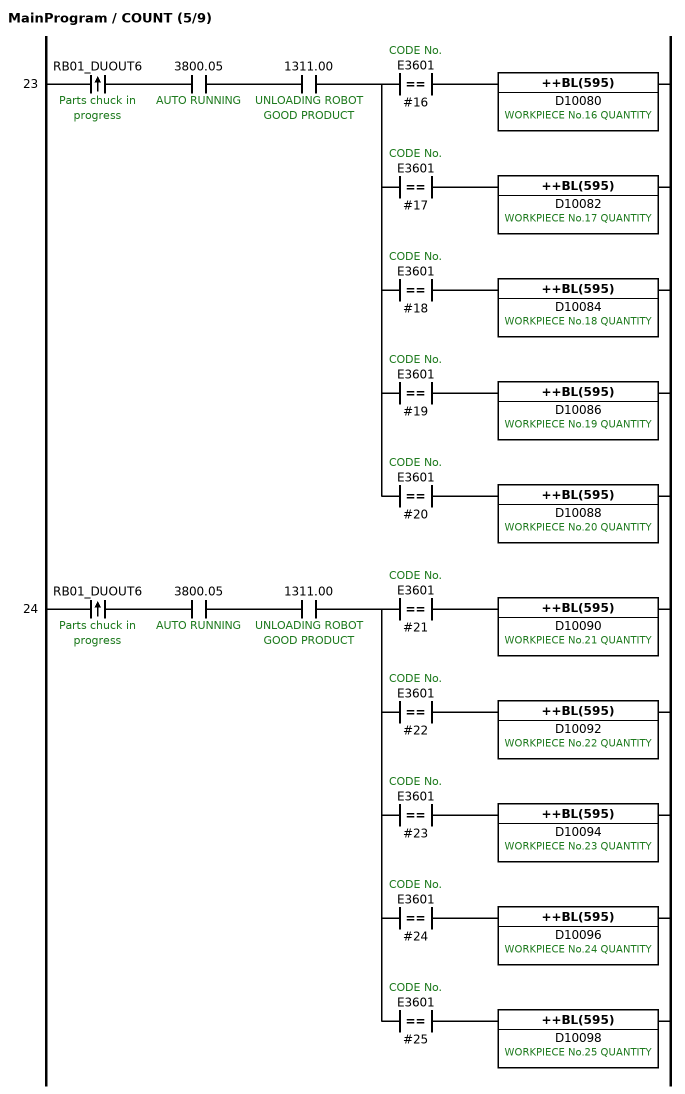
; [picture p144: MainProgram / COUNT, rungs 23-24]
; rung 23
@LD RB01_DUOUT6  ; Parts chuck in progress
AND 3800.05  ; AUTO RUNNING
AND 1311.00  ; UNLOADING ROBOT GOOD PRODUCT
OUT TR0
AND=(300) E3601 #16  ; CODE No.
++BL(595) D10080  ; WORKPIECE No.16 QUANTITY
LD TR0
AND=(300) E3601 #17  ; CODE No.
++BL(595) D10082  ; WORKPIECE No.17 QUANTITY
LD TR0
AND=(300) E3601 #18  ; CODE No.
++BL(595) D10084  ; WORKPIECE No.18 QUANTITY
LD TR0
AND=(300) E3601 #19  ; CODE No.
++BL(595) D10086  ; WORKPIECE No.19 QUANTITY
LD TR0
AND=(300) E3601 #20  ; CODE No.
++BL(595) D10088  ; WORKPIECE No.20 QUANTITY
; rung 24
@LD RB01_DUOUT6  ; Parts chuck in progress
AND 3800.05  ; AUTO RUNNING
AND 1311.00  ; UNLOADING ROBOT GOOD PRODUCT
OUT TR0
AND=(300) E3601 #21  ; CODE No.
++BL(595) D10090  ; WORKPIECE No.21 QUANTITY
LD TR0
AND=(300) E3601 #22  ; CODE No.
++BL(595) D10092  ; WORKPIECE No.22 QUANTITY
LD TR0
AND=(300) E3601 #23  ; CODE No.
++BL(595) D10094  ; WORKPIECE No.23 QUANTITY
LD TR0
AND=(300) E3601 #24  ; CODE No.
++BL(595) D10096  ; WORKPIECE No.24 QUANTITY
LD TR0
AND=(300) E3601 #25  ; CODE No.
++BL(595) D10098  ; WORKPIECE No.25 QUANTITY

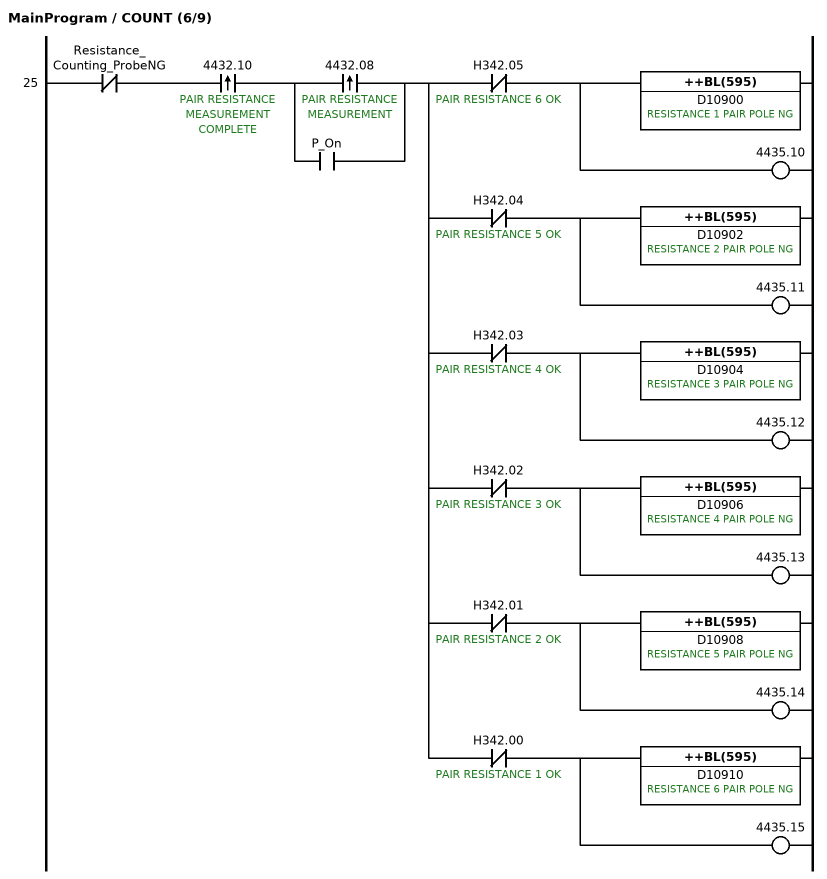
; rung 25
LDNOT Resistance_Counting_ProbeNG
@AND 4432.10  ; PAIR RESISTANCE MEASUREMENT COMPLETE
@LD 4432.08  ; PAIR RESISTANCE MEASUREMENT
OR P_On
ANDLD
OUT TR0
ANDNOT H342.05  ; PAIR RESISTANCE 6 OK
++BL(595) D10900  ; RESISTANCE 1 PAIR POLE NG
OUT 4435.10
LD TR0
ANDNOT H342.04  ; PAIR RESISTANCE 5 OK
++BL(595) D10902  ; RESISTANCE 2 PAIR POLE NG
OUT 4435.11
LD TR0
ANDNOT H342.03  ; PAIR RESISTANCE 4 OK
++BL(595) D10904  ; RESISTANCE 3 PAIR POLE NG
OUT 4435.12
LD TR0
ANDNOT H342.02  ; PAIR RESISTANCE 3 OK
++BL(595) D10906  ; RESISTANCE 4 PAIR POLE NG
OUT 4435.13
LD TR0
ANDNOT H342.01  ; PAIR RESISTANCE 2 OK
++BL(595) D10908  ; RESISTANCE 5 PAIR POLE NG
OUT 4435.14
LD TR0
ANDNOT H342.00  ; PAIR RESISTANCE 1 OK
++BL(595) D10910  ; RESISTANCE 6 PAIR POLE NG
OUT 4435.15

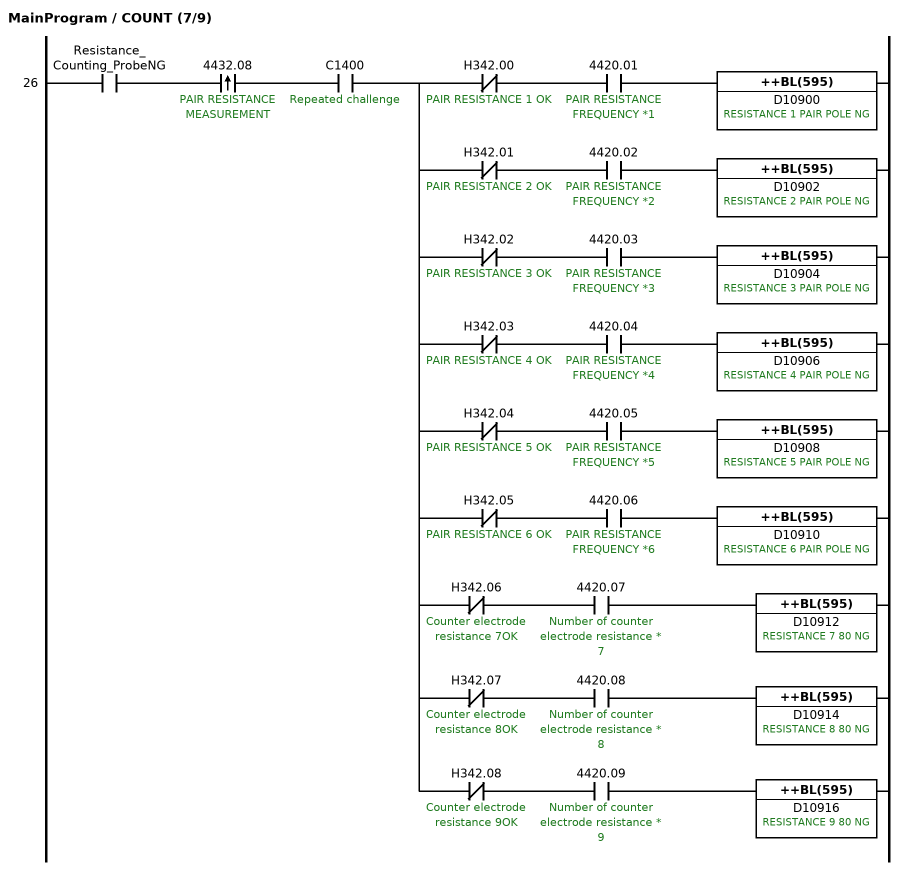
; rung 26
LD Resistance_Counting_ProbeNG
@AND 4432.08  ; PAIR RESISTANCE MEASUREMENT
AND C1400  ; Repeated challenge
OUT TR0
ANDNOT H342.00  ; PAIR RESISTANCE 1 OK
AND 4420.01  ; PAIR RESISTANCE FREQUENCY *1
++BL(595) D10900  ; RESISTANCE 1 PAIR POLE NG
LD TR0
ANDNOT H342.01  ; PAIR RESISTANCE 2 OK
AND 4420.02  ; PAIR RESISTANCE FREQUENCY *2
++BL(595) D10902  ; RESISTANCE 2 PAIR POLE NG
LD TR0
ANDNOT H342.02  ; PAIR RESISTANCE 3 OK
AND 4420.03  ; PAIR RESISTANCE FREQUENCY *3
++BL(595) D10904  ; RESISTANCE 3 PAIR POLE NG
LD TR0
ANDNOT H342.03  ; PAIR RESISTANCE 4 OK
AND 4420.04  ; PAIR RESISTANCE FREQUENCY *4
++BL(595) D10906  ; RESISTANCE 4 PAIR POLE NG
LD TR0
ANDNOT H342.04  ; PAIR RESISTANCE 5 OK
AND 4420.05  ; PAIR RESISTANCE FREQUENCY *5
++BL(595) D10908  ; RESISTANCE 5 PAIR POLE NG
LD TR0
ANDNOT H342.05  ; PAIR RESISTANCE 6 OK
AND 4420.06  ; PAIR RESISTANCE FREQUENCY *6
++BL(595) D10910  ; RESISTANCE 6 PAIR POLE NG
LD TR0
ANDNOT H342.06  ; Counter electrode resistance 7OK
AND 4420.07  ; Number of counter electrode resistance * 7
++BL(595) D10912  ; RESISTANCE 7 80 NG
LD TR0
ANDNOT H342.07  ; Counter electrode resistance 8OK
AND 4420.08  ; Number of counter electrode resistance * 8
++BL(595) D10914  ; RESISTANCE 8 80 NG
LD TR0
ANDNOT H342.08  ; Counter electrode resistance 9OK
AND 4420.09  ; Number of counter electrode resistance * 9
++BL(595) D10916  ; RESISTANCE 9 80 NG

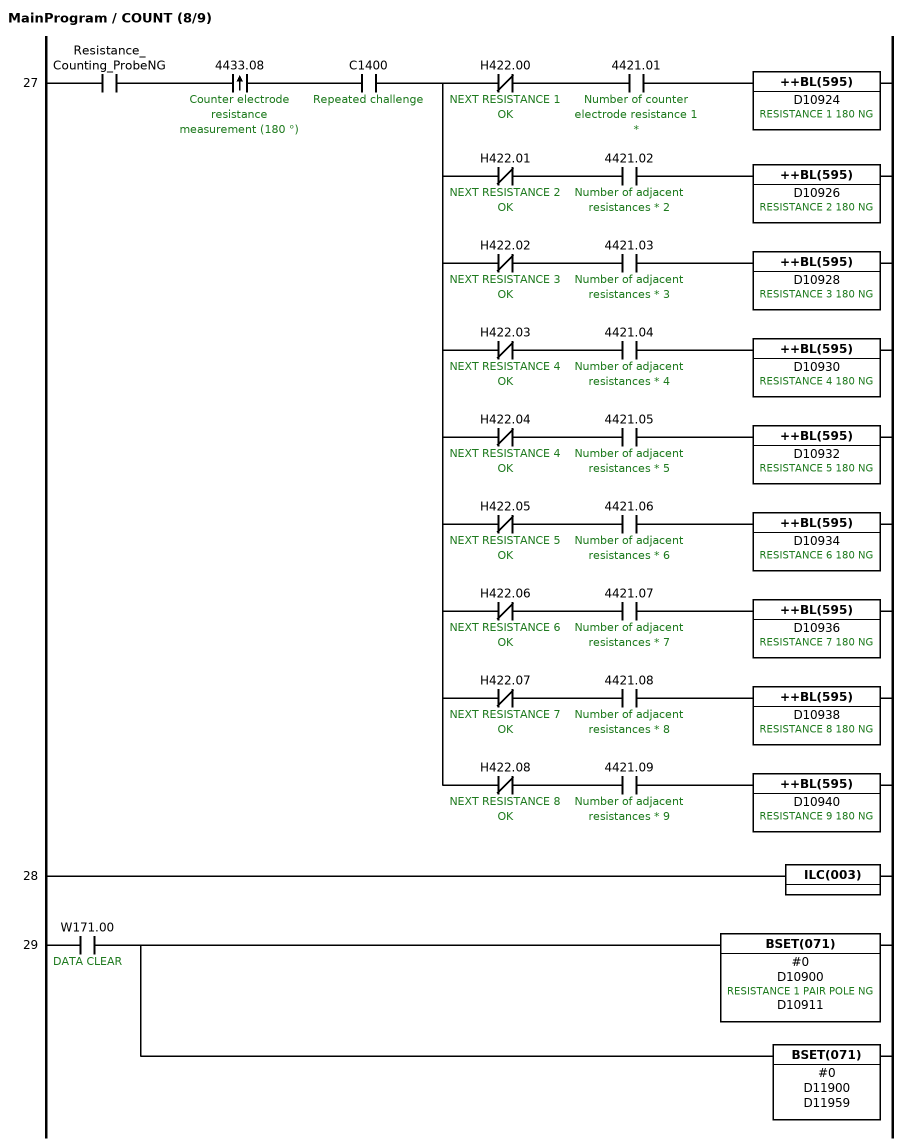
; rung 27
LD Resistance_Counting_ProbeNG
@AND 4433.08  ; Counter electrode resistance measurement (180 °)
AND C1400  ; Repeated challenge
OUT TR0
ANDNOT H422.00  ; NEXT RESISTANCE 1 OK
AND 4421.01  ; Number of counter electrode resistance 1 *
++BL(595) D10924  ; RESISTANCE 1 180 NG
LD TR0
ANDNOT H422.01  ; NEXT RESISTANCE 2 OK
AND 4421.02  ; Number of adjacent resistances * 2
++BL(595) D10926  ; RESISTANCE 2 180 NG
LD TR0
ANDNOT H422.02  ; NEXT RESISTANCE 3 OK
AND 4421.03  ; Number of adjacent resistances * 3
++BL(595) D10928  ; RESISTANCE 3 180 NG
LD TR0
ANDNOT H422.03  ; NEXT RESISTANCE 4 OK
AND 4421.04  ; Number of adjacent resistances * 4
++BL(595) D10930  ; RESISTANCE 4 180 NG
LD TR0
ANDNOT H422.04  ; NEXT RESISTANCE 4 OK
AND 4421.05  ; Number of adjacent resistances * 5
++BL(595) D10932  ; RESISTANCE 5 180 NG
LD TR0
ANDNOT H422.05  ; NEXT RESISTANCE 5 OK
AND 4421.06  ; Number of adjacent resistances * 6
++BL(595) D10934  ; RESISTANCE 6 180 NG
LD TR0
ANDNOT H422.06  ; NEXT RESISTANCE 6 OK
AND 4421.07  ; Number of adjacent resistances * 7
++BL(595) D10936  ; RESISTANCE 7 180 NG
LD TR0
ANDNOT H422.07  ; NEXT RESISTANCE 7 OK
AND 4421.08  ; Number of adjacent resistances * 8
++BL(595) D10938  ; RESISTANCE 8 180 NG
LD TR0
ANDNOT H422.08  ; NEXT RESISTANCE 8 OK
AND 4421.09  ; Number of adjacent resistances * 9
++BL(595) D10940  ; RESISTANCE 9 180 NG
; rung 28
ILC(003)
; rung 29
LD W171.00  ; DATA CLEAR
BSET(071) #0 D10900 D10911  ; RESISTANCE 1 PAIR POLE NG
BSET(071) #0 D11900 D11959

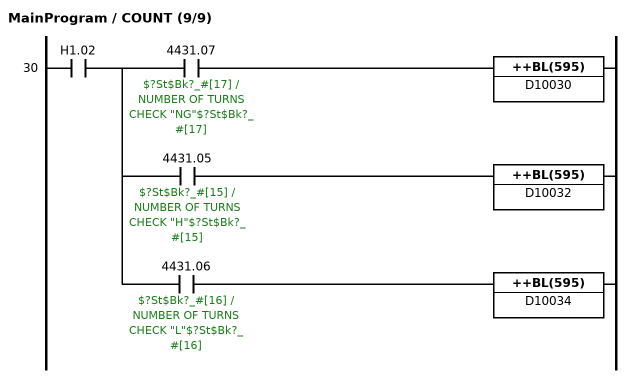
; rung 30
LD H1.02
OUT TR0
AND 4431.07  ; $?St$Bk?_#[17] / NUMBER OF TURNS CHECK "NG"$?St$Bk?_#[17]
++BL(595) D10030
LD TR0
AND 4431.05  ; $?St$Bk?_#[15] / NUMBER OF TURNS CHECK "H"$?St$Bk?_#[15]
++BL(595) D10032
LD TR0
AND 4431.06  ; $?St$Bk?_#[16] / NUMBER OF TURNS CHECK "L"$?St$Bk?_#[16]
++BL(595) D10034

### Section CONVEYOR

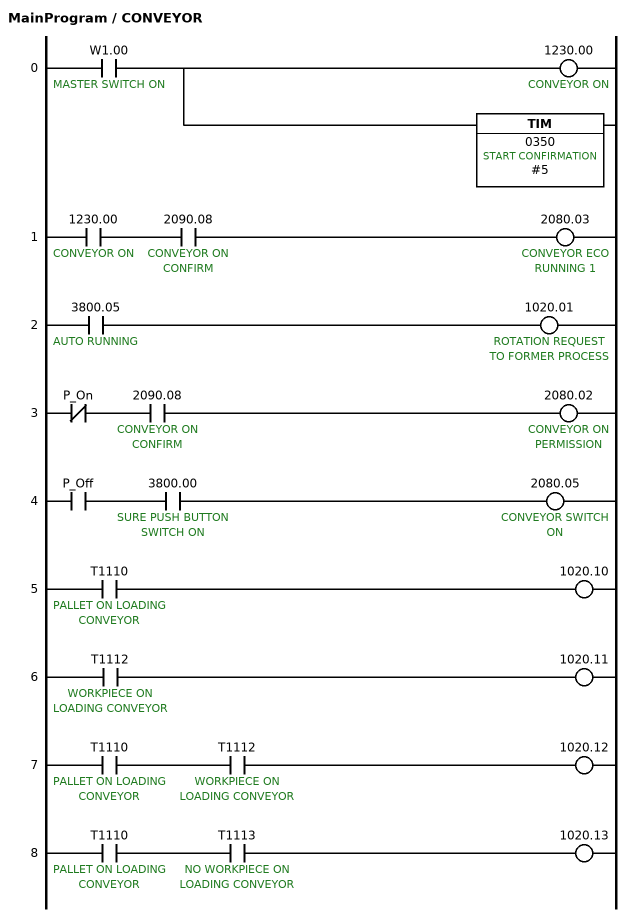
; rung 0
LD W1.00  ; MASTER SWITCH ON
OUT 1230.00  ; CONVEYOR ON
TIM 0350 #5  ; START CONFIRMATION
; rung 1
LD 1230.00  ; CONVEYOR ON
AND 2090.08  ; CONVEYOR ON CONFIRM
OUT 2080.03  ; CONVEYOR ECO RUNNING 1
; rung 2
LD 3800.05  ; AUTO RUNNING
OUT 1020.01  ; ROTATION REQUEST TO FORMER PROCESS
; rung 3
LDNOT P_On
AND 2090.08  ; CONVEYOR ON CONFIRM
OUT 2080.02  ; CONVEYOR ON PERMISSION
; rung 4
LD P_Off
AND 3800.00  ; SURE PUSH BUTTON SWITCH ON
OUT 2080.05  ; CONVEYOR SWITCH ON
; rung 5
LD T1110  ; PALLET ON LOADING CONVEYOR
OUT 1020.10
; rung 6
LD T1112  ; WORKPIECE ON LOADING CONVEYOR
OUT 1020.11
; rung 7
LD T1110  ; PALLET ON LOADING CONVEYOR
AND T1112  ; WORKPIECE ON LOADING CONVEYOR
OUT 1020.12
; rung 8
LD T1110  ; PALLET ON LOADING CONVEYOR
AND T1113  ; NO WORKPIECE ON LOADING CONVEYOR
OUT 1020.13

### Section ANALOG_INPUT

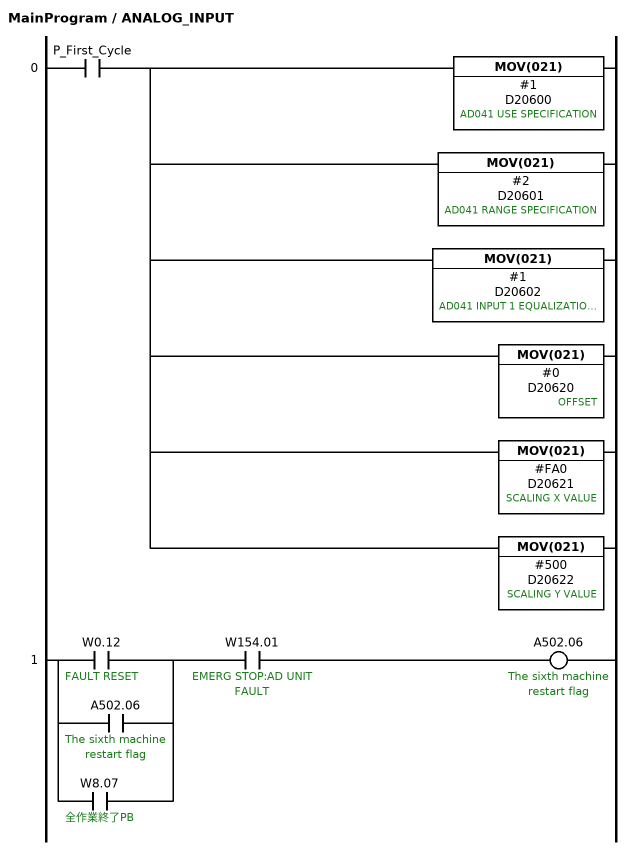
; rung 0
LD P_First_Cycle
MOV(021) #1 D20600  ; AD041 USE SPECIFICATION
MOV(021) #2 D20601  ; AD041 RANGE SPECIFICATION
MOV(021) #1 D20602  ; AD041 INPUT 1 EQUALIZATION PROCESSING
MOV(021) #0 D20620  ; OFFSET
MOV(021) #FA0 D20621  ; SCALING X VALUE
MOV(021) #500 D20622  ; SCALING Y VALUE
; rung 1
LD W0.12  ; FAULT RESET
OR A502.06  ; The sixth machine restart flag
OR W8.07  ; 全作業終了PB
AND W154.01  ; EMERG STOP:AD UNIT FAULT
OUT A502.06  ; The sixth machine restart flag

### Section Master_Check

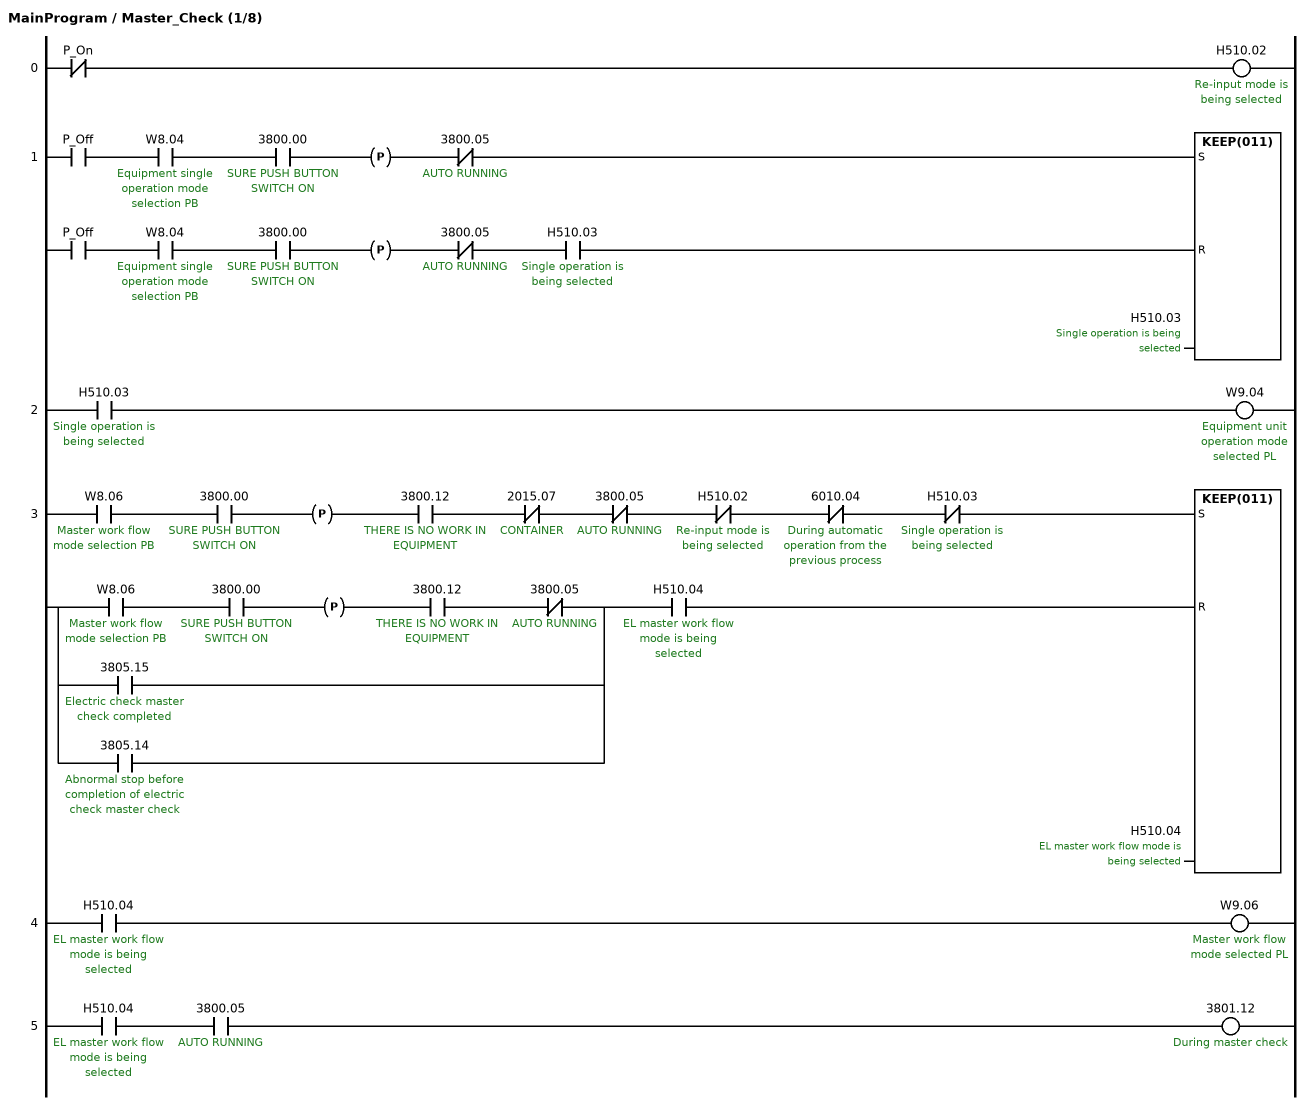
; rung 0
LDNOT P_On
OUT H510.02  ; Re-input mode is being selected
; rung 1
LD P_Off
AND W8.04  ; Equipment single operation mode selection PB
AND 3800.00  ; SURE PUSH BUTTON SWITCH ON
UP(521)
ANDNOT 3800.05  ; AUTO RUNNING
LD P_Off
AND W8.04  ; Equipment single operation mode selection PB
AND 3800.00  ; SURE PUSH BUTTON SWITCH ON
UP(521)
ANDNOT 3800.05  ; AUTO RUNNING
AND H510.03  ; Single operation is being selected
KEEP(011) H510.03  ; Single operation is being selected
; rung 2
LD H510.03  ; Single operation is being selected
OUT W9.04  ; Equipment unit operation mode selected PL
; rung 3
LD W8.06  ; Master work flow mode selection PB
AND 3800.00  ; SURE PUSH BUTTON SWITCH ON
UP(521)
AND 3800.12  ; THERE IS NO WORK IN EQUIPMENT
ANDNOT 2015.07  ; CONTAINER
ANDNOT 3800.05  ; AUTO RUNNING
ANDNOT H510.02  ; Re-input mode is being selected
ANDNOT 6010.04  ; During automatic operation from the previous process
ANDNOT H510.03  ; Single operation is being selected
LD W8.06  ; Master work flow mode selection PB
AND 3800.00  ; SURE PUSH BUTTON SWITCH ON
UP(521)
AND 3800.12  ; THERE IS NO WORK IN EQUIPMENT
ANDNOT 3800.05  ; AUTO RUNNING
OR 3805.15  ; Electric check master check completed
OR 3805.14  ; Abnormal stop before completion of electric check master check
AND H510.04  ; EL master work flow mode is being selected
KEEP(011) H510.04  ; EL master work flow mode is being selected
; rung 4
LD H510.04  ; EL master work flow mode is being selected
OUT W9.06  ; Master work flow mode selected PL
; rung 5
LD H510.04  ; EL master work flow mode is being selected
AND 3800.05  ; AUTO RUNNING
OUT 3801.12  ; During master check

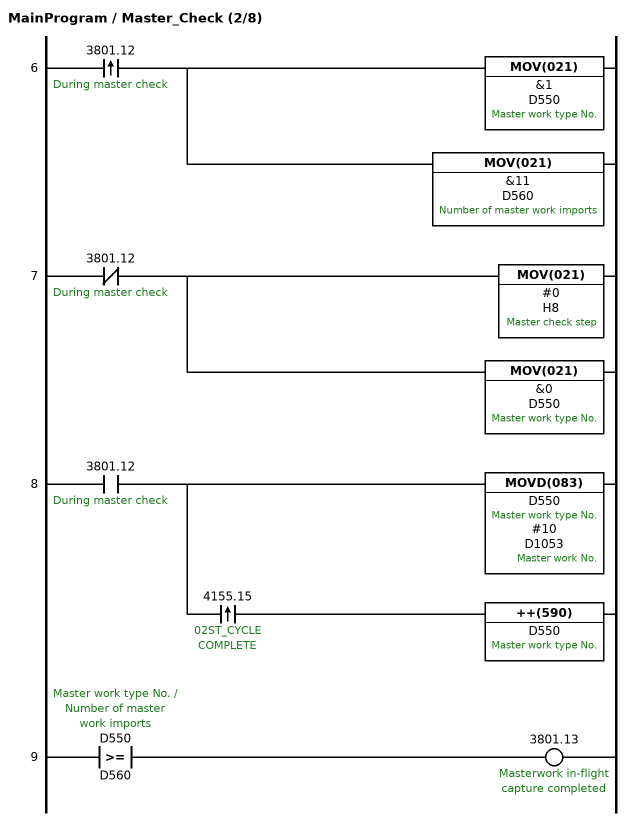
; rung 6
@LD 3801.12  ; During master check
MOV(021) &1 D550  ; Master work type No.
MOV(021) &11 D560  ; Number of master work imports
; rung 7
LDNOT 3801.12  ; During master check
MOV(021) #0 H8  ; Master check step
MOV(021) &0 D550  ; Master work type No.
; rung 8
LD 3801.12  ; During master check
MOVD(083) D550 #10 D1053  ; Master work type No., Master work No.
@AND 4155.15  ; 02ST_CYCLE COMPLETE
++(590) D550  ; Master work type No.
; rung 9
LD>=(325) D550 D560  ; Master work type No., Number of master work imports
OUT 3801.13  ; Masterwork in-flight capture completed

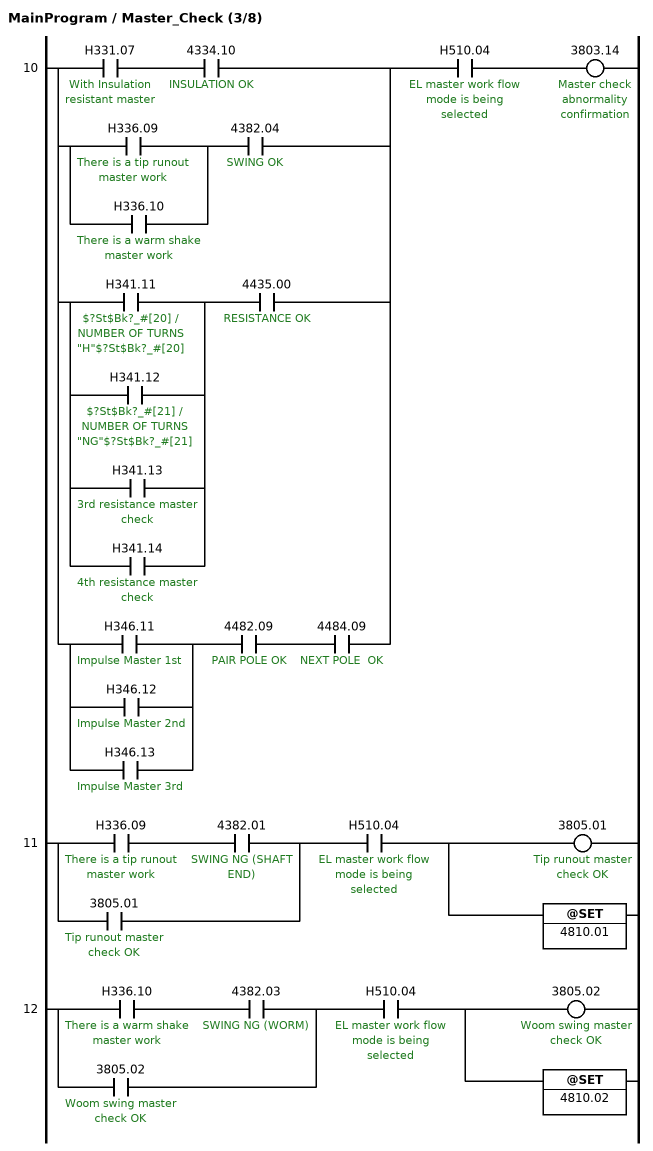
; rung 10
LD H331.07  ; With Insulation resistant master
AND 4334.10  ; INSULATION OK
LD H336.09  ; There is a tip runout master work
OR H336.10  ; There is a warm shake master work
AND 4382.04  ; SWING OK
ORLD
LD H341.11  ; $?St$Bk?_#[20] / NUMBER OF TURNS "H"$?St$Bk?_#[20]
OR H341.12  ; $?St$Bk?_#[21] / NUMBER OF TURNS "NG"$?St$Bk?_#[21]
OR H341.13  ; 3rd resistance master check
OR H341.14  ; 4th resistance master check
AND 4435.00  ; RESISTANCE OK
ORLD
LD H346.11  ; Impulse Master 1st
OR H346.12  ; Impulse Master 2nd
OR H346.13  ; Impulse Master 3rd
AND 4482.09  ; PAIR POLE OK
AND 4484.09  ; NEXT POLE  OK
ORLD
AND H510.04  ; EL master work flow mode is being selected
OUT 3803.14  ; Master check abnormality confirmation
; rung 11
LD H336.09  ; There is a tip runout master work
AND 4382.01  ; SWING NG (SHAFT END)
OR 3805.01  ; Tip runout master check OK
AND H510.04  ; EL master work flow mode is being selected
OUT 3805.01  ; Tip runout master check OK
@SET 4810.01
; rung 12
LD H336.10  ; There is a warm shake master work
AND 4382.03  ; SWING NG (WORM)
OR 3805.02  ; Woom swing master check OK
AND H510.04  ; EL master work flow mode is being selected
OUT 3805.02  ; Woom swing master check OK
@SET 4810.02

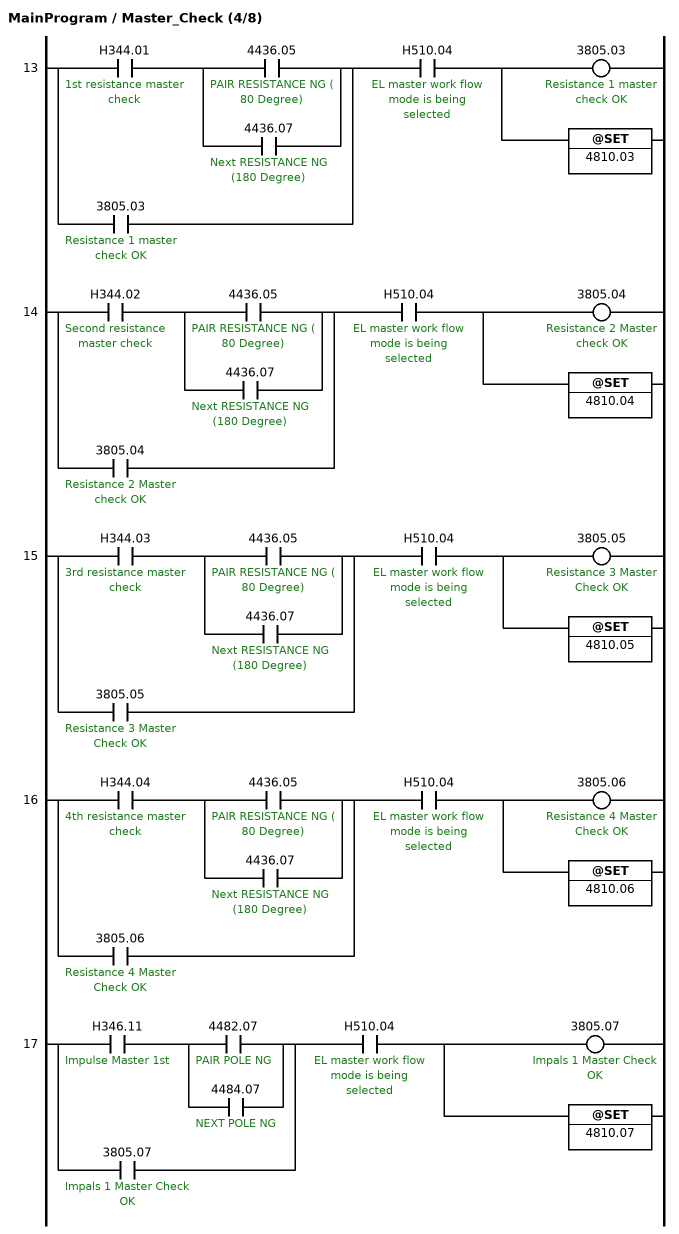
; rung 13
LD H344.01  ; 1st resistance master check
LD 4436.05  ; PAIR RESISTANCE NG ( 80 Degree)
OR 4436.07  ; Next RESISTANCE NG (180 Degree)
ANDLD
OR 3805.03  ; Resistance 1 master check OK
AND H510.04  ; EL master work flow mode is being selected
OUT 3805.03  ; Resistance 1 master check OK
@SET 4810.03
; rung 14
LD H344.02  ; Second resistance master check
LD 4436.05  ; PAIR RESISTANCE NG ( 80 Degree)
OR 4436.07  ; Next RESISTANCE NG (180 Degree)
ANDLD
OR 3805.04  ; Resistance 2 Master check OK
AND H510.04  ; EL master work flow mode is being selected
OUT 3805.04  ; Resistance 2 Master check OK
@SET 4810.04
; rung 15
LD H344.03  ; 3rd resistance master check
LD 4436.05  ; PAIR RESISTANCE NG ( 80 Degree)
OR 4436.07  ; Next RESISTANCE NG (180 Degree)
ANDLD
OR 3805.05  ; Resistance 3 Master Check OK
AND H510.04  ; EL master work flow mode is being selected
OUT 3805.05  ; Resistance 3 Master Check OK
@SET 4810.05
; rung 16
LD H344.04  ; 4th resistance master check
LD 4436.05  ; PAIR RESISTANCE NG ( 80 Degree)
OR 4436.07  ; Next RESISTANCE NG (180 Degree)
ANDLD
OR 3805.06  ; Resistance 4 Master Check OK
AND H510.04  ; EL master work flow mode is being selected
OUT 3805.06  ; Resistance 4 Master Check OK
@SET 4810.06
; rung 17
LD H346.11  ; Impulse Master 1st
LD 4482.07  ; PAIR POLE NG
OR 4484.07  ; NEXT POLE NG
ANDLD
OR 3805.07  ; Impals 1 Master Check OK
AND H510.04  ; EL master work flow mode is being selected
OUT 3805.07  ; Impals 1 Master Check OK
@SET 4810.07

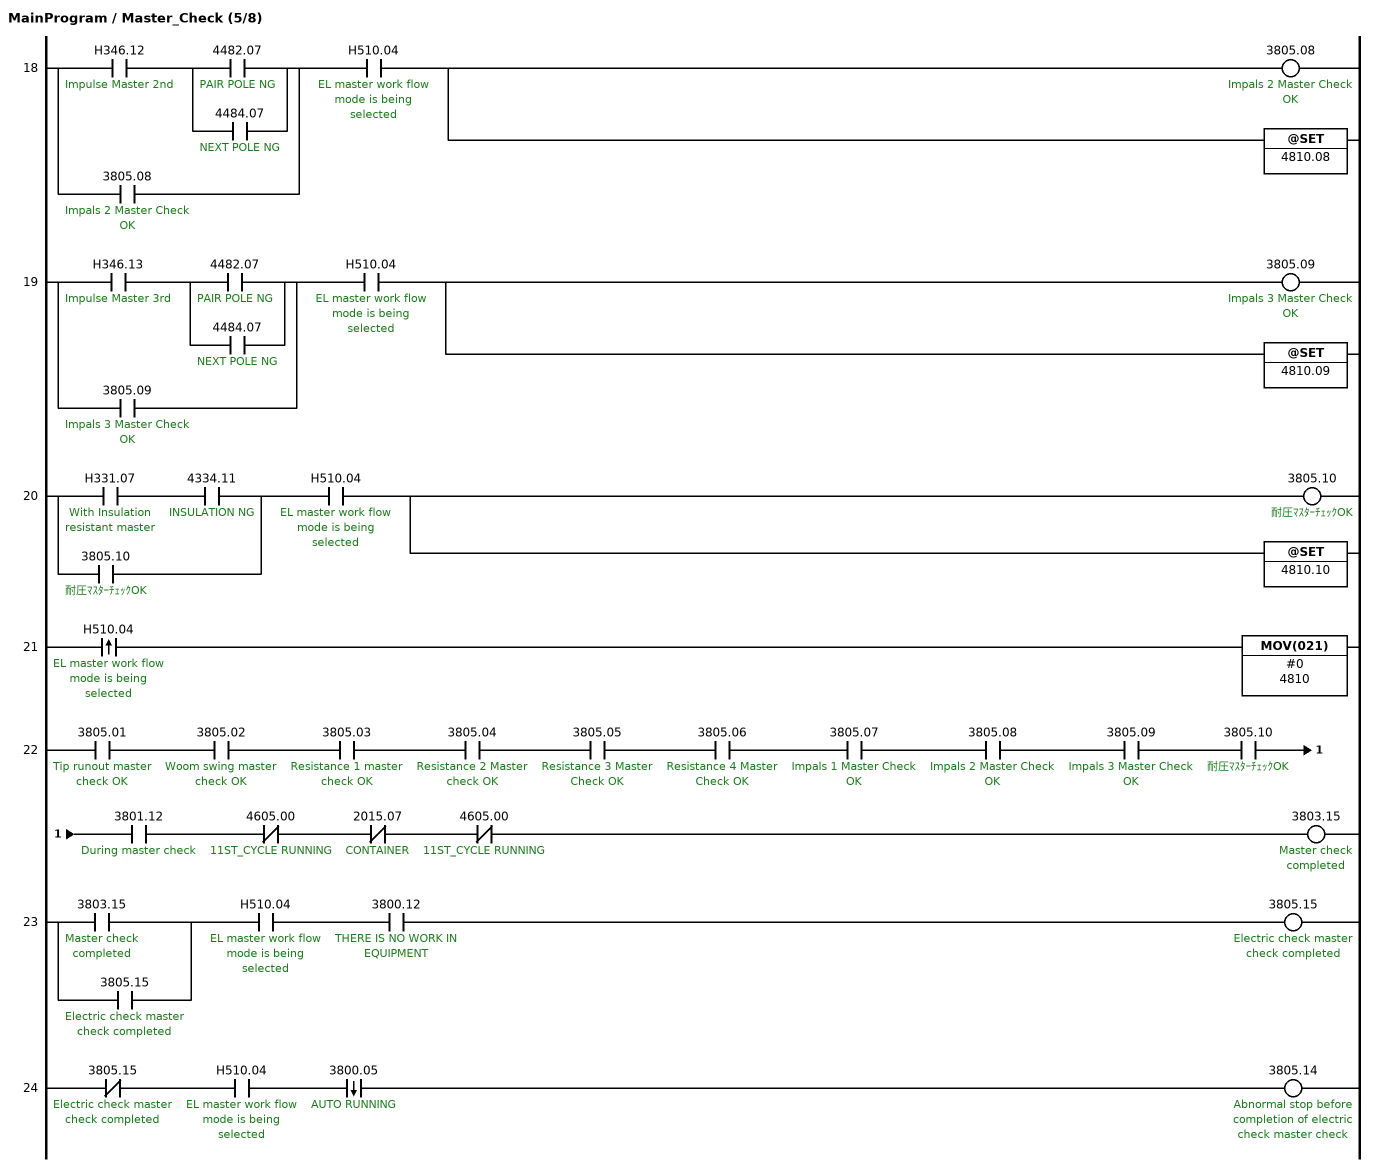
; rung 18
LD H346.12  ; Impulse Master 2nd
LD 4482.07  ; PAIR POLE NG
OR 4484.07  ; NEXT POLE NG
ANDLD
OR 3805.08  ; Impals 2 Master Check OK
AND H510.04  ; EL master work flow mode is being selected
OUT 3805.08  ; Impals 2 Master Check OK
@SET 4810.08
; rung 19
LD H346.13  ; Impulse Master 3rd
LD 4482.07  ; PAIR POLE NG
OR 4484.07  ; NEXT POLE NG
ANDLD
OR 3805.09  ; Impals 3 Master Check OK
AND H510.04  ; EL master work flow mode is being selected
OUT 3805.09  ; Impals 3 Master Check OK
@SET 4810.09
; rung 20
LD H331.07  ; With Insulation resistant master
AND 4334.11  ; INSULATION NG
OR 3805.10  ; 耐圧ﾏｽﾀｰﾁｪｯｸOK
AND H510.04  ; EL master work flow mode is being selected
OUT 3805.10  ; 耐圧ﾏｽﾀｰﾁｪｯｸOK
@SET 4810.10
; rung 21
@LD H510.04  ; EL master work flow mode is being selected
MOV(021) #0 4810
; rung 22
LD 3805.01  ; Tip runout master check OK
AND 3805.02  ; Woom swing master check OK
AND 3805.03  ; Resistance 1 master check OK
AND 3805.04  ; Resistance 2 Master check OK
AND 3805.05  ; Resistance 3 Master Check OK
AND 3805.06  ; Resistance 4 Master Check OK
AND 3805.07  ; Impals 1 Master Check OK
AND 3805.08  ; Impals 2 Master Check OK
AND 3805.09  ; Impals 3 Master Check OK
AND 3805.10  ; 耐圧ﾏｽﾀｰﾁｪｯｸOK
AND 3801.12  ; During master check
ANDNOT 4605.00  ; 11ST_CYCLE RUNNING
ANDNOT 2015.07  ; CONTAINER
ANDNOT 4605.00  ; 11ST_CYCLE RUNNING
OUT 3803.15  ; Master check completed
; rung 23
LD 3803.15  ; Master check completed
OR 3805.15  ; Electric check master check completed
AND H510.04  ; EL master work flow mode is being selected
AND 3800.12  ; THERE IS NO WORK IN EQUIPMENT
OUT 3805.15  ; Electric check master check completed
; rung 24
LDNOT 3805.15  ; Electric check master check completed
AND H510.04  ; EL master work flow mode is being selected
%AND 3800.05  ; AUTO RUNNING
OUT 3805.14  ; Abnormal stop before completion of electric check master check

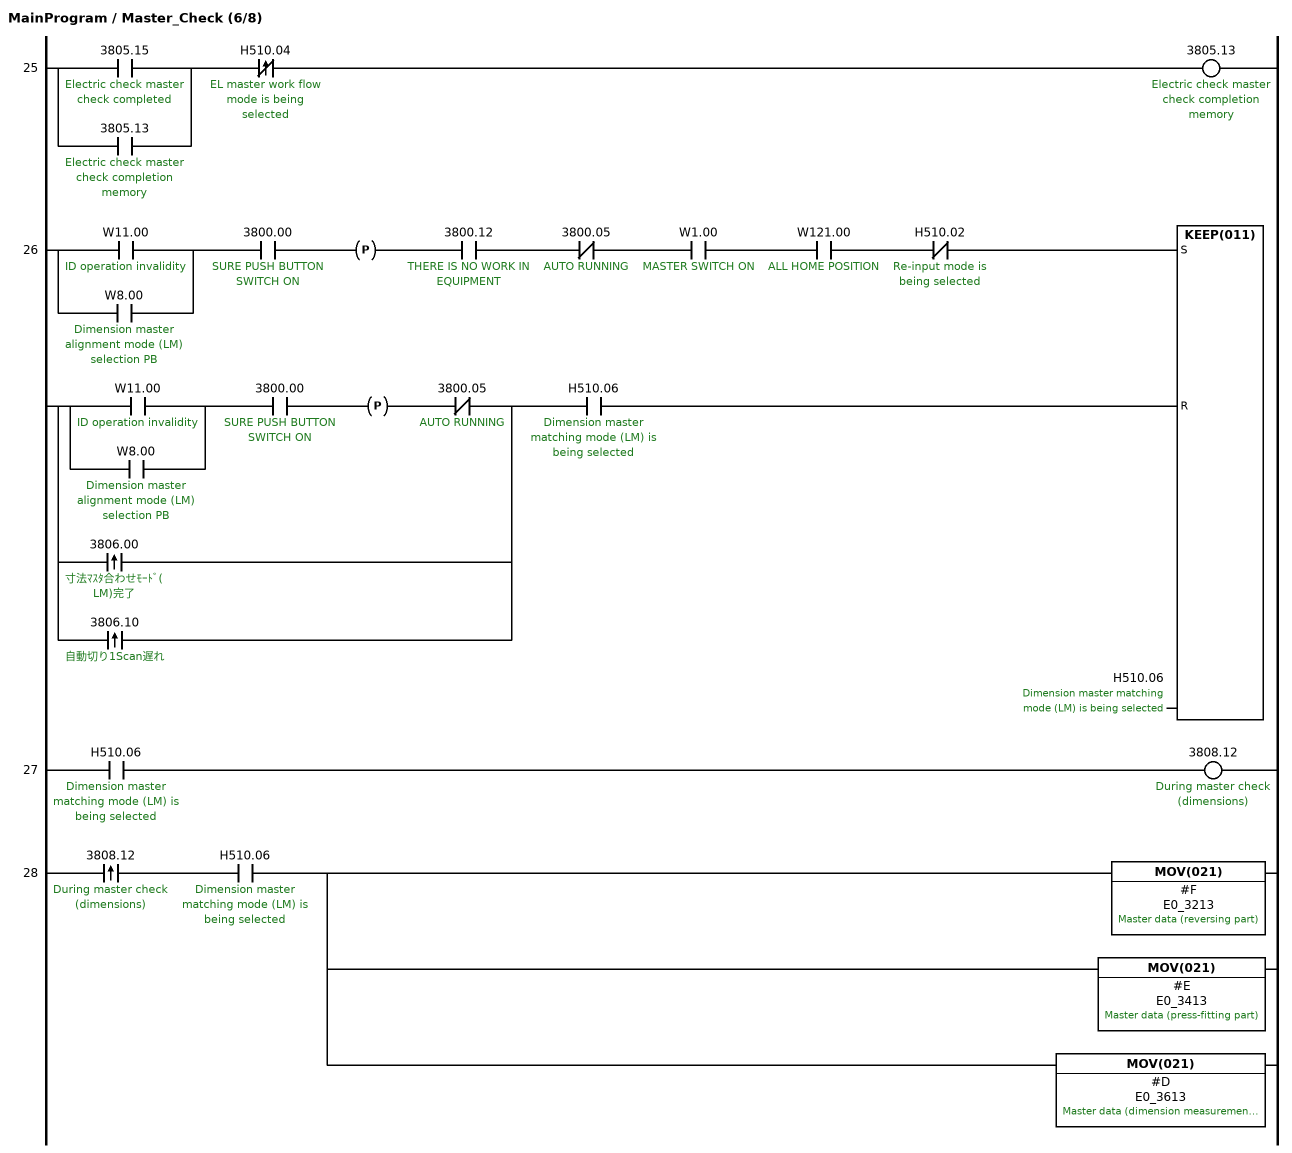
; rung 25
LD 3805.15  ; Electric check master check completed
OR 3805.13  ; Electric check master check completion memory
@ANDNOT H510.04  ; EL master work flow mode is being selected
OUT 3805.13  ; Electric check master check completion memory
; rung 26
LD W11.00  ; ID operation invalidity
OR W8.00  ; Dimension master alignment mode (LM) selection PB
AND 3800.00  ; SURE PUSH BUTTON SWITCH ON
UP(521)
AND 3800.12  ; THERE IS NO WORK IN EQUIPMENT
ANDNOT 3800.05  ; AUTO RUNNING
AND W1.00  ; MASTER SWITCH ON
AND W121.00  ; ALL HOME POSITION
ANDNOT H510.02  ; Re-input mode is being selected
LD W11.00  ; ID operation invalidity
OR W8.00  ; Dimension master alignment mode (LM) selection PB
AND 3800.00  ; SURE PUSH BUTTON SWITCH ON
UP(521)
ANDNOT 3800.05  ; AUTO RUNNING
@OR 3806.00  ; 寸法ﾏｽﾀ合わせﾓｰﾄﾞ(LM)完了
@OR 3806.10  ; 自動切り1Scan遅れ
AND H510.06  ; Dimension master matching mode (LM) is being selected
KEEP(011) H510.06  ; Dimension master matching mode (LM) is being selected
; rung 27
LD H510.06  ; Dimension master matching mode (LM) is being selected
OUT 3808.12  ; During master check (dimensions)
; rung 28
@LD 3808.12  ; During master check (dimensions)
AND H510.06  ; Dimension master matching mode (LM) is being selected
MOV(021) #F E0_3213  ; Master data (reversing part)
MOV(021) #E E0_3413  ; Master data (press-fitting part)
MOV(021) #D E0_3613  ; Master data (dimension measurement unit)

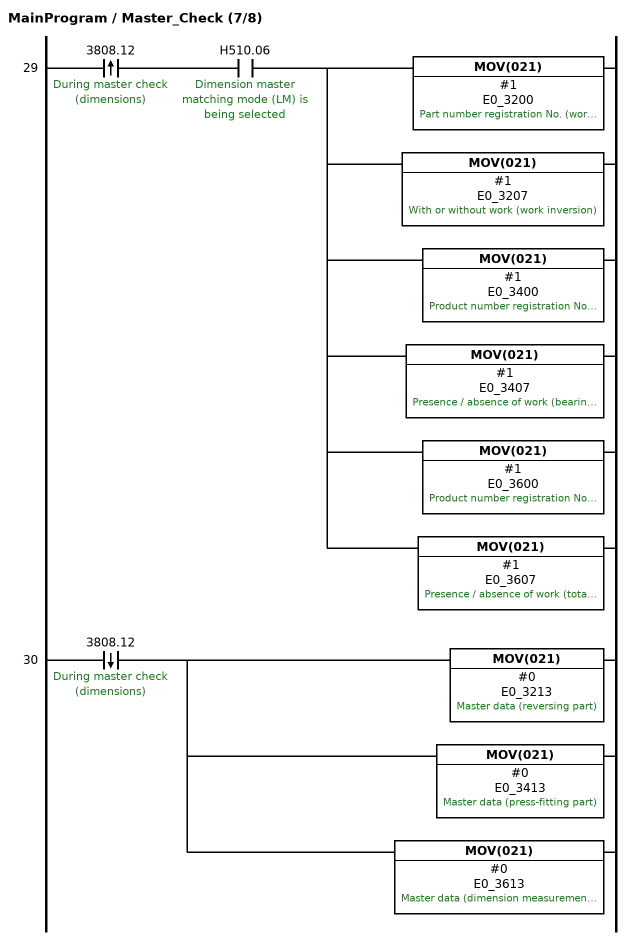
; rung 29
@LD 3808.12  ; During master check (dimensions)
AND H510.06  ; Dimension master matching mode (LM) is being selected
MOV(021) #1 E0_3200  ; Part number registration No. (work reversal)
MOV(021) #1 E0_3207  ; With or without work (work inversion)
MOV(021) #1 E0_3400  ; Product number registration No. (bearing press-fitting)
MOV(021) #1 E0_3407  ; Presence / absence of work (bearing press-fitting)
MOV(021) #1 E0_3600  ; Product number registration No. (total length measurement)
MOV(021) #1 E0_3607  ; Presence / absence of work (total length measurement)
; rung 30
%LD 3808.12  ; During master check (dimensions)
MOV(021) #0 E0_3213  ; Master data (reversing part)
MOV(021) #0 E0_3413  ; Master data (press-fitting part)
MOV(021) #0 E0_3613  ; Master data (dimension measurement unit)

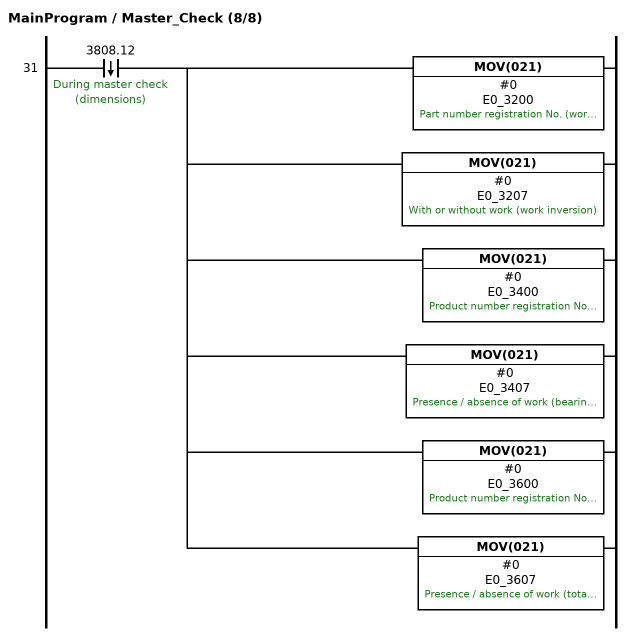
; rung 31
%LD 3808.12  ; During master check (dimensions)
MOV(021) #0 E0_3200  ; Part number registration No. (work reversal)
MOV(021) #0 E0_3207  ; With or without work (work inversion)
MOV(021) #0 E0_3400  ; Product number registration No. (bearing press-fitting)
MOV(021) #0 E0_3407  ; Presence / absence of work (bearing press-fitting)
MOV(021) #0 E0_3600  ; Product number registration No. (total length measurement)
MOV(021) #0 E0_3607  ; Presence / absence of work (total length measurement)

### Section HIGH_SPEED_COUNTER

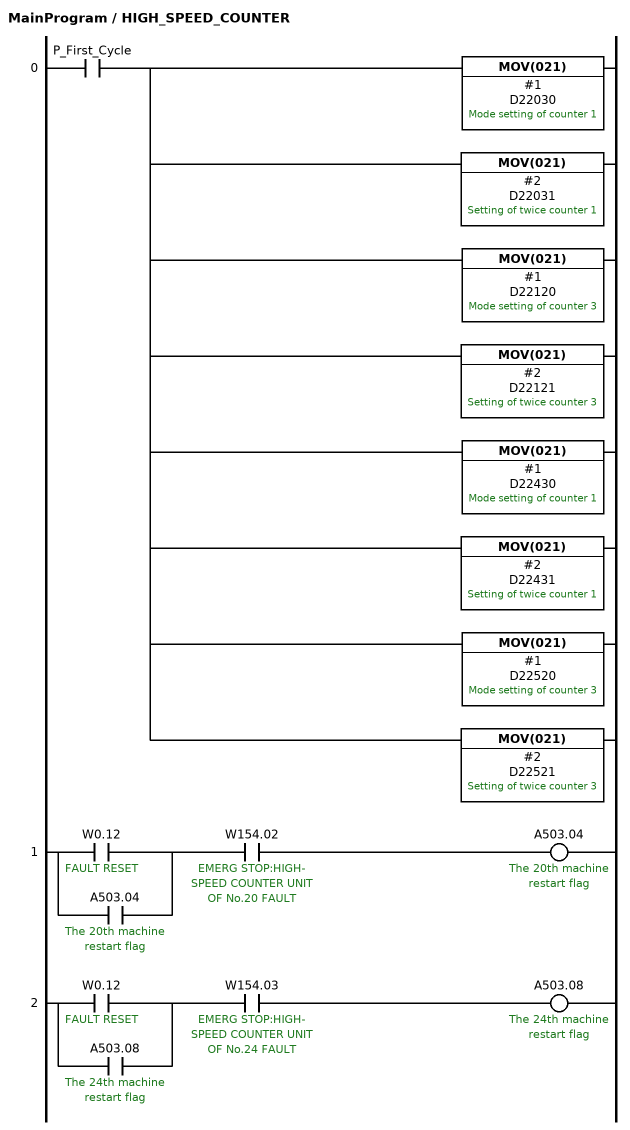
; rung 0
LD P_First_Cycle
MOV(021) #1 D22030  ; Mode setting of counter 1
MOV(021) #2 D22031  ; Setting of twice counter 1
MOV(021) #1 D22120  ; Mode setting of counter 3
MOV(021) #2 D22121  ; Setting of twice counter 3
MOV(021) #1 D22430  ; Mode setting of counter 1
MOV(021) #2 D22431  ; Setting of twice counter 1
MOV(021) #1 D22520  ; Mode setting of counter 3
MOV(021) #2 D22521  ; Setting of twice counter 3
; rung 1
LD W0.12  ; FAULT RESET
OR A503.04  ; The 20th machine restart flag
AND W154.02  ; EMERG STOP:HIGH-SPEED COUNTER UNIT OF No.20 FAULT
OUT A503.04  ; The 20th machine restart flag
; rung 2
LD W0.12  ; FAULT RESET
OR A503.08  ; The 24th machine restart flag
AND W154.03  ; EMERG STOP:HIGH-SPEED COUNTER UNIT OF No.24 FAULT
OUT A503.08  ; The 24th machine restart flag

### Section DATA_SAVING

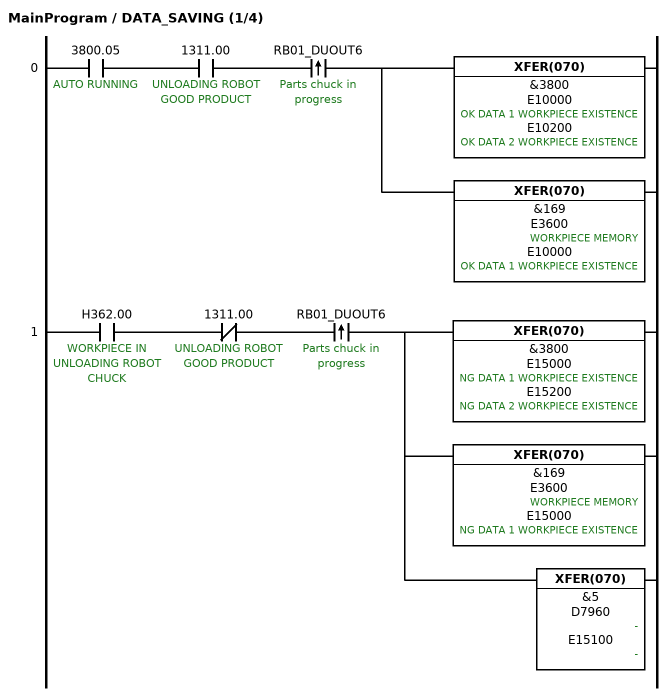
; rung 0
LD 3800.05  ; AUTO RUNNING
AND 1311.00  ; UNLOADING ROBOT GOOD PRODUCT
@AND RB01_DUOUT6  ; Parts chuck in progress
XFER(070) &3800 E10000 E10200  ; OK DATA 1 WORKPIECE EXISTENCE, OK DATA 2 WORKPIECE EXISTENCE
XFER(070) &169 E3600 E10000  ; WORKPIECE MEMORY, OK DATA 1 WORKPIECE EXISTENCE
; rung 1
LD H362.00  ; WORKPIECE IN UNLOADING ROBOT CHUCK
ANDNOT 1311.00  ; UNLOADING ROBOT GOOD PRODUCT
@AND RB01_DUOUT6  ; Parts chuck in progress
XFER(070) &3800 E15000 E15200  ; NG DATA 1 WORKPIECE EXISTENCE, NG DATA 2 WORKPIECE EXISTENCE
XFER(070) &169 E3600 E15000  ; WORKPIECE MEMORY, NG DATA 1 WORKPIECE EXISTENCE
XFER(070) &5 D7960 E15100  ; -

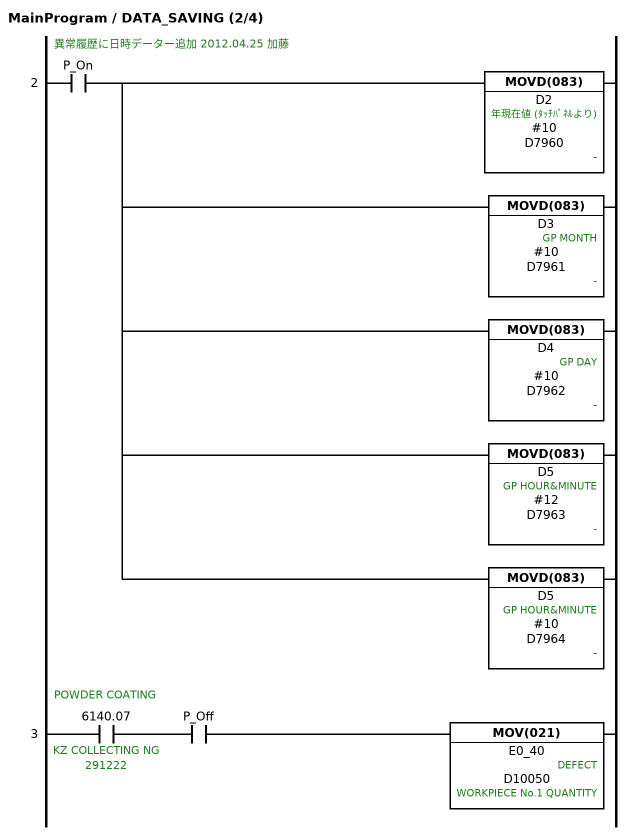
; rung 2: 異常履歴に日時データー追加 2012.04.25 加藤
LD P_On
MOVD(083) D2 #10 D7960  ; 年現在値 (ﾀｯﾁﾊﾟﾈﾙより), -
MOVD(083) D3 #10 D7961  ; GP MONTH, -
MOVD(083) D4 #10 D7962  ; GP DAY, -
MOVD(083) D5 #12 D7963  ; GP HOUR&MINUTE, -
MOVD(083) D5 #10 D7964  ; GP HOUR&MINUTE, -
; rung 3: POWDER COATING
LD 6140.07  ; KZ COLLECTING NG 291222
AND P_Off
MOV(021) E0_40 D10050  ; DEFECT, WORKPIECE No.1 QUANTITY

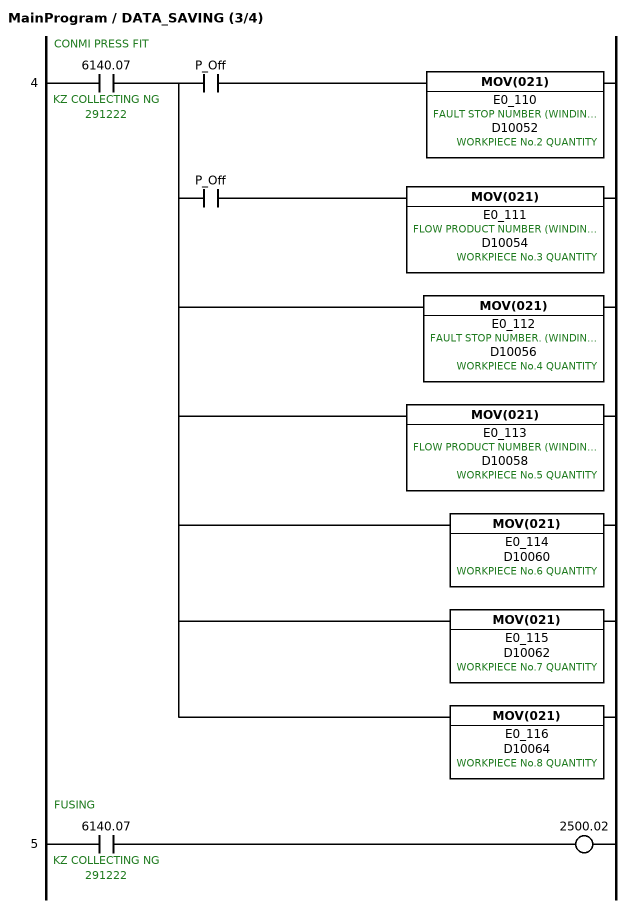
; rung 4: CONMI PRESS FIT
LD 6140.07  ; KZ COLLECTING NG 291222
OUT TR0
AND P_Off
MOV(021) E0_110 D10052  ; FAULT STOP NUMBER (WINDING No.1), WORKPIECE No.2 QUANTITY
LD TR0
AND P_Off
MOV(021) E0_111 D10054  ; FLOW PRODUCT NUMBER (WINDING No.1), WORKPIECE No.3 QUANTITY
LD TR0
MOV(021) E0_112 D10056  ; FAULT STOP NUMBER. (WINDING No.2), WORKPIECE No.4 QUANTITY
MOV(021) E0_113 D10058  ; FLOW PRODUCT NUMBER (WINDING No.2), WORKPIECE No.5 QUANTITY
MOV(021) E0_114 D10060  ; WORKPIECE No.6 QUANTITY
MOV(021) E0_115 D10062  ; WORKPIECE No.7 QUANTITY
MOV(021) E0_116 D10064  ; WORKPIECE No.8 QUANTITY
; rung 5: FUSING
LD 6140.07  ; KZ COLLECTING NG 291222
OUT 2500.02

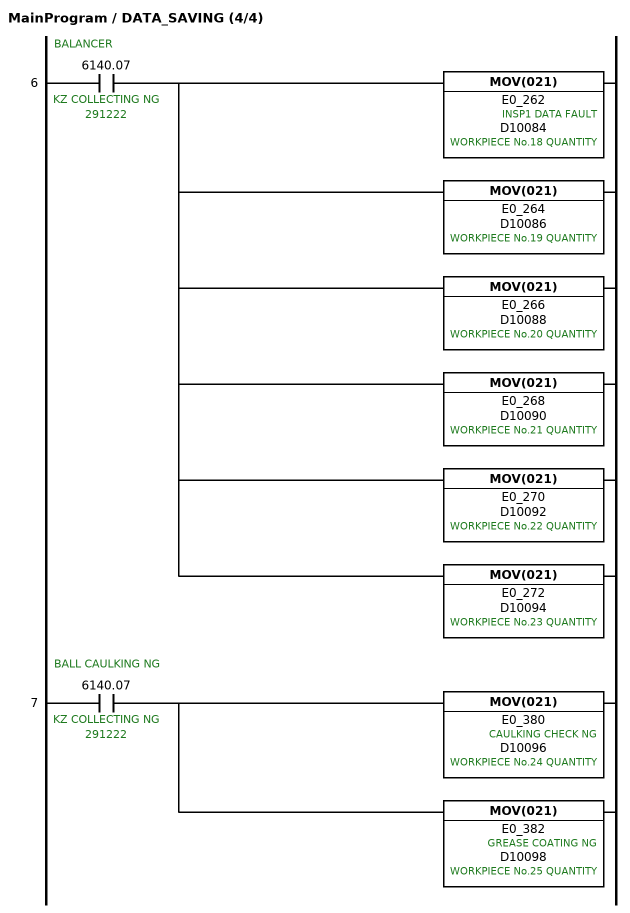
; rung 6: BALANCER
LD 6140.07  ; KZ COLLECTING NG 291222
MOV(021) E0_262 D10084  ; INSP1 DATA FAULT, WORKPIECE No.18 QUANTITY
MOV(021) E0_264 D10086  ; WORKPIECE No.19 QUANTITY
MOV(021) E0_266 D10088  ; WORKPIECE No.20 QUANTITY
MOV(021) E0_268 D10090  ; WORKPIECE No.21 QUANTITY
MOV(021) E0_270 D10092  ; WORKPIECE No.22 QUANTITY
MOV(021) E0_272 D10094  ; WORKPIECE No.23 QUANTITY
; rung 7: BALL CAULKING NG
LD 6140.07  ; KZ COLLECTING NG 291222
MOV(021) E0_380 D10096  ; CAULKING CHECK NG, WORKPIECE No.24 QUANTITY
MOV(021) E0_382 D10098  ; GREASE COATING NG, WORKPIECE No.25 QUANTITY

### Section DATA_HISTORY

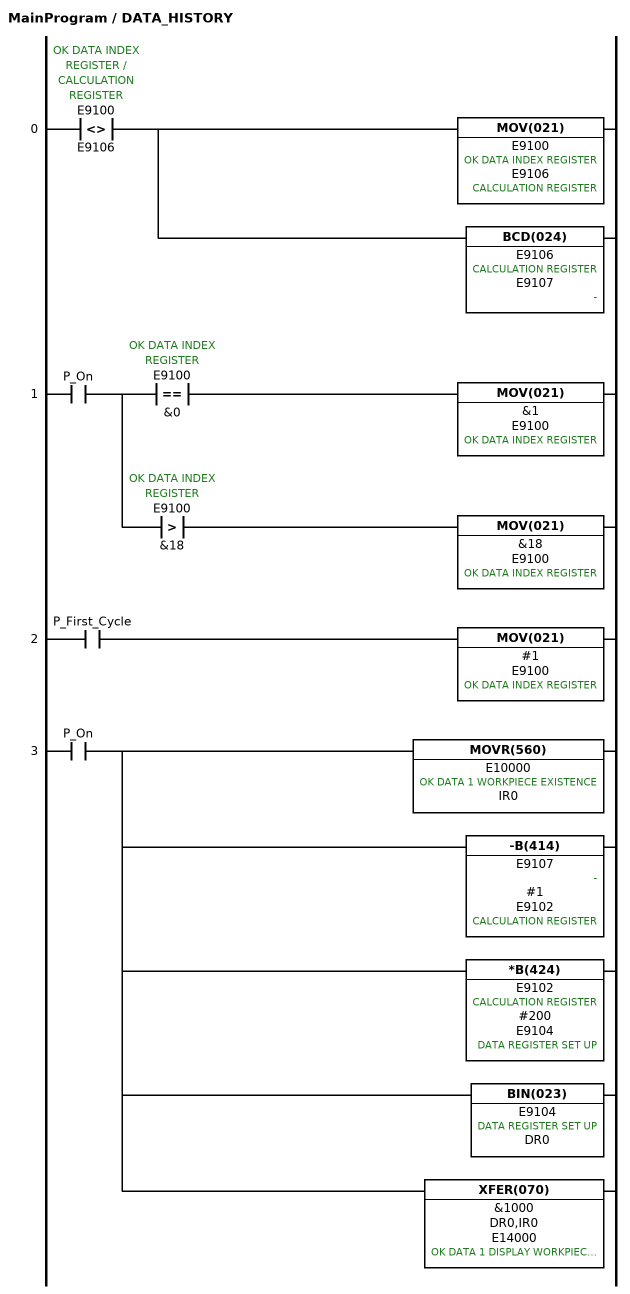
; rung 0
LD<>(305) E9100 E9106  ; OK DATA INDEX REGISTER, CALCULATION REGISTER
MOV(021) E9100 E9106  ; OK DATA INDEX REGISTER, CALCULATION REGISTER
BCD(024) E9106 E9107  ; CALCULATION REGISTER, -
; rung 1
LD P_On
OUT TR0
AND=(300) E9100 &0  ; OK DATA INDEX REGISTER
MOV(021) &1 E9100  ; OK DATA INDEX REGISTER
LD TR0
AND>(320) E9100 &18  ; OK DATA INDEX REGISTER
MOV(021) &18 E9100  ; OK DATA INDEX REGISTER
; rung 2
LD P_First_Cycle
MOV(021) #1 E9100  ; OK DATA INDEX REGISTER
; rung 3
LD P_On
MOVR(560) E10000 IR0  ; OK DATA 1 WORKPIECE EXISTENCE
-B(414) E9107 #1 E9102  ; -, CALCULATION REGISTER
*B(424) E9102 #200 E9104  ; CALCULATION REGISTER, DATA REGISTER SET UP
BIN(023) E9104 DR0  ; DATA REGISTER SET UP
XFER(070) &1000 DR0,IR0 E14000  ; OK DATA 1 DISPLAY WORKPIECE EXISTENCE

### Section DATA_HISTORY_2

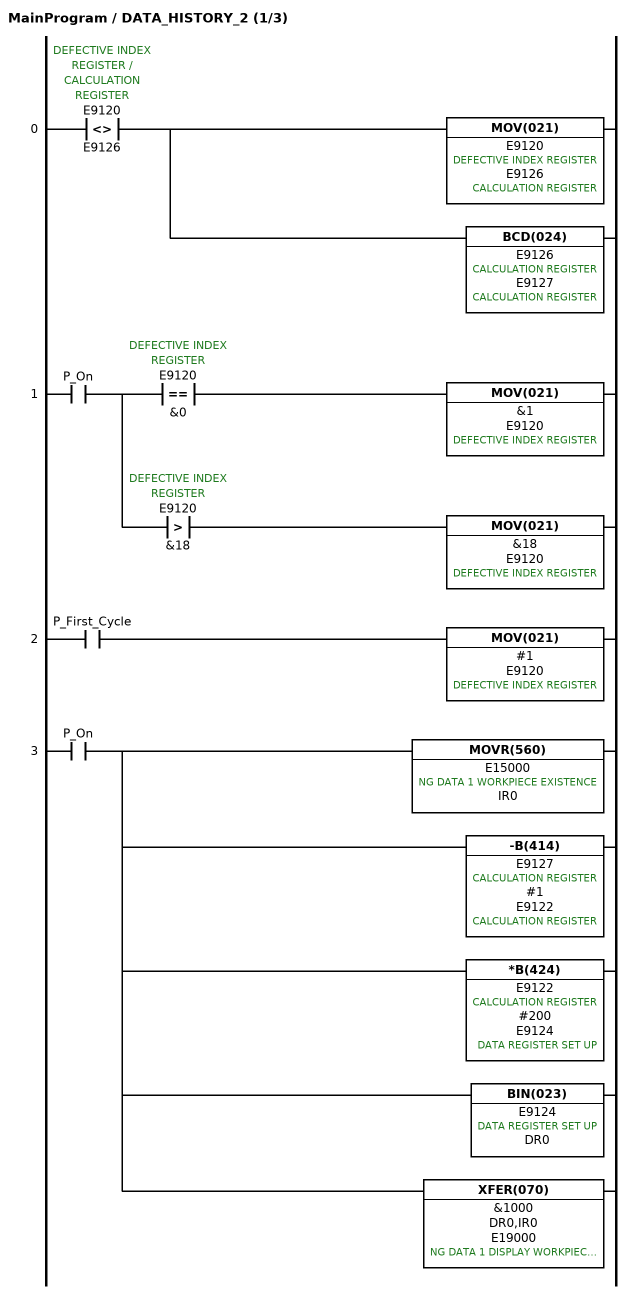
; rung 0
LD<>(305) E9120 E9126  ; DEFECTIVE INDEX REGISTER, CALCULATION REGISTER
MOV(021) E9120 E9126  ; DEFECTIVE INDEX REGISTER, CALCULATION REGISTER
BCD(024) E9126 E9127  ; CALCULATION REGISTER
; rung 1
LD P_On
OUT TR0
AND=(300) E9120 &0  ; DEFECTIVE INDEX REGISTER
MOV(021) &1 E9120  ; DEFECTIVE INDEX REGISTER
LD TR0
AND>(320) E9120 &18  ; DEFECTIVE INDEX REGISTER
MOV(021) &18 E9120  ; DEFECTIVE INDEX REGISTER
; rung 2
LD P_First_Cycle
MOV(021) #1 E9120  ; DEFECTIVE INDEX REGISTER
; rung 3
LD P_On
MOVR(560) E15000 IR0  ; NG DATA 1 WORKPIECE EXISTENCE
-B(414) E9127 #1 E9122  ; CALCULATION REGISTER
*B(424) E9122 #200 E9124  ; CALCULATION REGISTER, DATA REGISTER SET UP
BIN(023) E9124 DR0  ; DATA REGISTER SET UP
XFER(070) &1000 DR0,IR0 E19000  ; NG DATA 1 DISPLAY WORKPIECE EXISTENCE

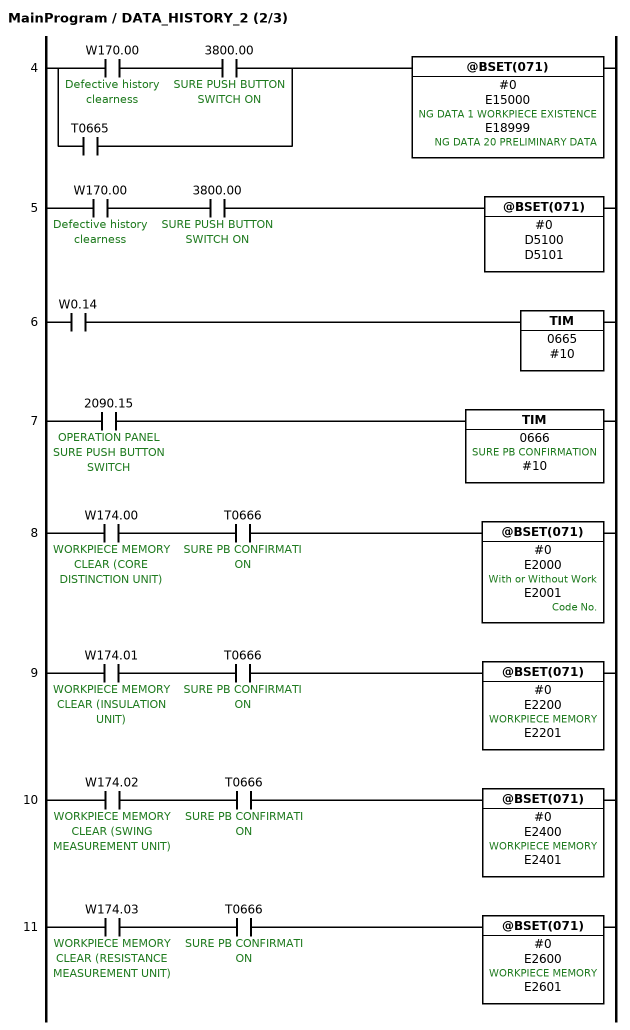
; rung 4
LD W170.00  ; Defective history clearness
AND 3800.00  ; SURE PUSH BUTTON SWITCH ON
OR T0665
@BSET(071) #0 E15000 E18999  ; NG DATA 1 WORKPIECE EXISTENCE, NG DATA 20 PRELIMINARY DATA
; rung 5
LD W170.00  ; Defective history clearness
AND 3800.00  ; SURE PUSH BUTTON SWITCH ON
@BSET(071) #0 D5100 D5101
; rung 6
LD W0.14
TIM 0665 #10
; rung 7
LD 2090.15  ; OPERATION PANEL SURE PUSH BUTTON SWITCH
TIM 0666 #10  ; SURE PB CONFIRMATION
; rung 8
LD W174.00  ; WORKPIECE MEMORY CLEAR (CORE DISTINCTION UNIT)
AND T0666  ; SURE PB CONFIRMATION
@BSET(071) #0 E2000 E2001  ; With or Without Work, Code No.
; rung 9
LD W174.01  ; WORKPIECE MEMORY CLEAR (INSULATION UNIT)
AND T0666  ; SURE PB CONFIRMATION
@BSET(071) #0 E2200 E2201  ; WORKPIECE MEMORY
; rung 10
LD W174.02  ; WORKPIECE MEMORY CLEAR (SWING MEASUREMENT UNIT)
AND T0666  ; SURE PB CONFIRMATION
@BSET(071) #0 E2400 E2401  ; WORKPIECE MEMORY
; rung 11
LD W174.03  ; WORKPIECE MEMORY CLEAR (RESISTANCE MEASUREMENT UNIT)
AND T0666  ; SURE PB CONFIRMATION
@BSET(071) #0 E2600 E2601  ; WORKPIECE MEMORY

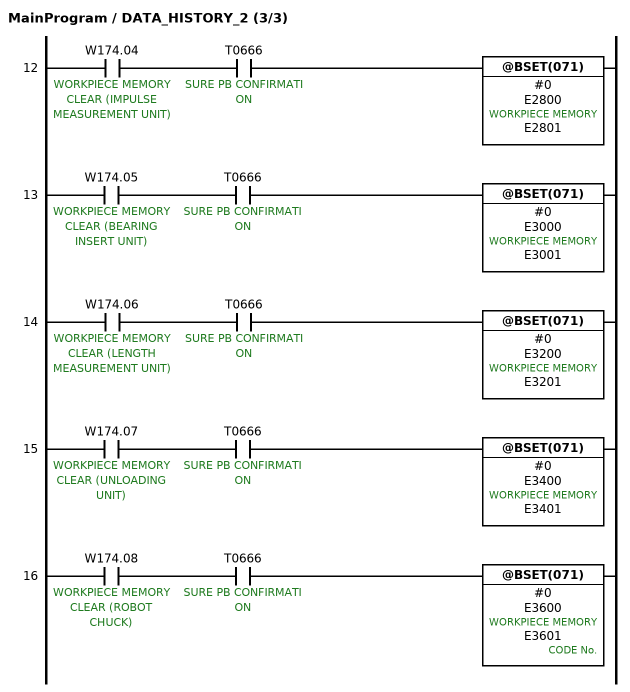
; rung 12
LD W174.04  ; WORKPIECE MEMORY CLEAR (IMPULSE MEASUREMENT UNIT)
AND T0666  ; SURE PB CONFIRMATION
@BSET(071) #0 E2800 E2801  ; WORKPIECE MEMORY
; rung 13
LD W174.05  ; WORKPIECE MEMORY CLEAR (BEARING INSERT UNIT)
AND T0666  ; SURE PB CONFIRMATION
@BSET(071) #0 E3000 E3001  ; WORKPIECE MEMORY
; rung 14
LD W174.06  ; WORKPIECE MEMORY CLEAR (LENGTH MEASUREMENT UNIT)
AND T0666  ; SURE PB CONFIRMATION
@BSET(071) #0 E3200 E3201  ; WORKPIECE MEMORY
; rung 15
LD W174.07  ; WORKPIECE MEMORY CLEAR (UNLOADING UNIT)
AND T0666  ; SURE PB CONFIRMATION
@BSET(071) #0 E3400 E3401  ; WORKPIECE MEMORY
; rung 16
LD W174.08  ; WORKPIECE MEMORY CLEAR (ROBOT CHUCK)
AND T0666  ; SURE PB CONFIRMATION
@BSET(071) #0 E3600 E3601  ; WORKPIECE MEMORY, CODE No.

### Section FAULT_STOP_HISTORY

